TYPE OPC_UA_REAL :
STRUCT
	NodeID				: ST_UANodeID;
	NodeHdl				: DWORD;
	SizeOfDataType		: UDINT;
	NodeAddInfo			: ST_UANodeAdditionalInfo;
	TargetVar			: POINTER TO REAL;
END_STRUCT
END_TYPE

(* stored: Version 1.1.0.1, ProductVersion 3.1.4024.9
   DUT OPC_UA_REAL: Id {1823d541-ff12-460e-8515-3a4a5d36e1b4} *)
